FUNCTION_BLOCK FB_FIS_oop IMPLEMENTS FuzzyInferenceSystem
VAR_INPUT
END_VAR
VAR_OUTPUT
END_VAR
VAR
END_VAR

END_FUNCTION_BLOCK

(* stored: Version 1.1.0.1, ProductVersion 3.1.4024.6
   POU FB_FIS_oop: Id {ea7a488c-96fc-40ed-9c89-6520d1adaaf5}, SpecialFunc None *)
